// TIA Portal V20 export
DATA_BLOCK "DB_Digital_Inputs"   // DB1
{ S7_Optimized_Access := 'TRUE' }
// stored: MemoryReserve 100
   VAR
      Button_Start_Approve : Bool;
      Digital_Input_1 : Bool;
      Digital_Input_2 : Bool;
      Digital_Input_3 : Bool;
      Digital_Input_4 : Bool;
      Digital_Input_5 : Bool;
   END_VAR
BEGIN
END_DATA_BLOCK
